KUKA KRL program: Rack_Verde_V.src, Rack_Verde_V.dat

--- Rack_Verde_V.src ---
&ACCESS RVO1
&REL 3
&COMMENT SECUENCIA RACK VERDE
&PARAM EDITMASK = *
&PARAM TEMPLATE = C:\KRC\Roboter\Template\vorgabe
DEF Rack_Verde_V( )
;FOLD INI;%{PE}
  ;FOLD BASISTECH INI
    GLOBAL INTERRUPT DECL 3 WHEN $STOPMESS==TRUE DO IR_STOPM ( )
    INTERRUPT ON 3
    BAS (#INITMOV,0 )
  ;ENDFOLD (BASISTECH INI)
;FOLD SPOTTECH INI
USERSPOT(#INIT)
;ENDFOLD (SPOTTECH INI)
;FOLD GRIPPERTECH INI
USER_GRP(0,DUMMY,DUMMY,GDEFAULT)
;ENDFOLD (GRIPPERTECH INI)
  ;FOLD USER INI
    ;Make your modifications here

  ;ENDFOLD (USER INI)
;ENDFOLD (INI)
;################################################
; PROYECTO: MAFELEC PLANTA DE BATERIAS
; ROBOT: 121_R1
; PROGRAMA: SECUENCIA DE TRABAJO ROBOT RACK VERDE
;           CON SISTEMA DE VISION SELECCIONADA
; CREADO POR: Un amigo en Balay(zaisor robotics)
; FECHA: 23-NOVIEMBRE-2022
; MODIFICADO POR:
; FECHA MODIFICACION: 10-ENERO-2023
;################################################

;FOLD PTP HOME Vel=100 % DEFAULT;%{PE}%R 8.3.48,%MKUKATPBASIS,%CMOVE,%VPTP,%P 1:PTP, 2:HOME, 3:, 5:100, 7:DEFAULT
$BWDSTART=FALSE
PDAT_ACT=PDEFAULT
FDAT_ACT=FHOME
BAS(#PTP_PARAMS,100)
$H_POS=XHOME
PTP XHOME
;ENDFOLD
$out[61]=false
FINALIZA_VERDE=FALSE
SELECT_NEXT=FALSE

Rack_Verde_Inpicker ()

IF (SELECT_NEXT==FALSE) AND (FINALIZA_VERDE==FALSE) THEN

;FOLD PTP POS_Wait_Verde_ST121 Vel=100 % H Tool[9]:T_Gripper1_Vacio Base[0];%{PE}%R 8.3.48,%MKUKATPBASIS,%CMOVE,%VPTP,%P 1:PTP, 2:POS_Wait_Verde_ST121, 3:, 5:100, 7:H
$BWDSTART=FALSE
PDAT_ACT=PH
FDAT_ACT=FPOS_Wait_Verde_ST121
BAS(#PTP_PARAMS,100)
PTP XPOS_Wait_Verde_ST121
;ENDFOLD

;ESPERA AREA 3 (ENTRADA COGER BATERIA EN ST121)
WAIT FOR I_ARDY_3
O_AREL_3=FALSE

IF (I_ST121_INSPECCION==TRUE) THEN
Rack_Verde_CogerST121I ()
ELSE
Rack_Verde_CogerST121N ()
ENDIF

Rack_Verde_Dejar()
ENDIF
$out[61]=true
FINALIZA_VERDE=FALSE
SELECT_NEXT=FALSE

;FOLD PTP HOME Vel=100 % DEFAULT;%{PE}%R 8.3.48,%MKUKATPBASIS,%CMOVE,%VPTP,%P 1:PTP, 2:HOME, 3:, 5:100, 7:DEFAULT
$BWDSTART=FALSE
PDAT_ACT=PDEFAULT
FDAT_ACT=FHOME
BAS(#PTP_PARAMS,100)
$H_POS=XHOME
PTP XHOME
;ENDFOLD
END

--- Rack_Verde_V.dat ---
&ACCESS RVO1
&REL 3
&COMMENT SECUENCIA RACK VERDE
&PARAM EDITMASK = *
&PARAM TEMPLATE = C:\KRC\Roboter\Template\vorgabe
DEFDAT  Rack_Verde_V
;FOLD EXTERNAL DECLARATIONS;%{PE}%MKUKATPBASIS,%CEXT,%VCOMMON,%P
;FOLD GRIPPERTECH EXT
EXT  H50 (INT  :IN,INT  :IN,INT  :IN,GRP_TYP  :IN )
;ENDFOLD (GRIPPERTECH EXT)
;FOLD SPOTTECH EXT
EXT  USERSPOT (S_COMMAND  :IN,SPOT_TYPE  :IN )
;ENDFOLD (SPOTTECH EXT)
;FOLD BASISTECH EXT;%{PE}%MKUKATPBASIS,%CEXT,%VEXT,%P
EXT  BAS (BAS_COMMAND  :IN,REAL  :IN )
DECL INT SUCCESS
;ENDFOLD (BASISTECH EXT)
;FOLD USER EXT;%{E}%MKUKATPUSER,%CEXT,%VEXT,%P
;Make your modifications here

;ENDFOLD (USER EXT)
;ENDFOLD (EXTERNAL DECLARATIONS)
DECL PDAT PH={VEL 100.000,ACC 100.000,APO_DIST 100.000,APO_MODE #CDIS,GEAR_JERK 50.0000,EXAX_IGN 0}
DECL E6POS XPOS_Wait_Verde_ST121={X 1606.70789,Y -354.796814,Z 1944.22656,A 1.33749425,B -32.3921471,C 179.037674,S 2,T 42,E1 0.0,E2 0.0,E3 0.0,E4 0.0,E5 0.0,E6 0.0}
DECL FDAT FPOS_Wait_Verde_ST121={TOOL_NO 9,BASE_NO 0,IPO_FRAME #BASE,POINT2[] " ",TQ_STATE FALSE}
ENDDAT
